// TIA Portal V19 export
TYPE "C501_VAR_HYK_TYPIC"
   STRUCT
      DEU { ExternalAccessible := 'False'; ExternalVisible := 'False'; ExternalWritable := 'False'} : USInt;   // De hydrantkast in de verkeerskoker is geopend
      OBS { ExternalAccessible := 'False'; ExternalVisible := 'False'; ExternalWritable := 'False'} : USInt;   // Observeerbaarheid
   END_STRUCT;
END_TYPE
